// TIA Portal V21 export
FUNCTION "xwaxwadfawd" : Void   // FC6, LAD
{ S7_Optimized_Access := 'TRUE' }
// stored: SetENOAutomatically false
BEGIN
END_FUNCTION
